// LS Electric XG5000 project: 주차설비
// PLC LSPLC
// module base 0 slot 0: 입출력 모듈:XBC-DN/DP64H (DC 24V 입력, 트랜지스터 출력 64점 (싱크출력/소스출력))

PROGRAM NewProgram (task: 스캔 프로그램)

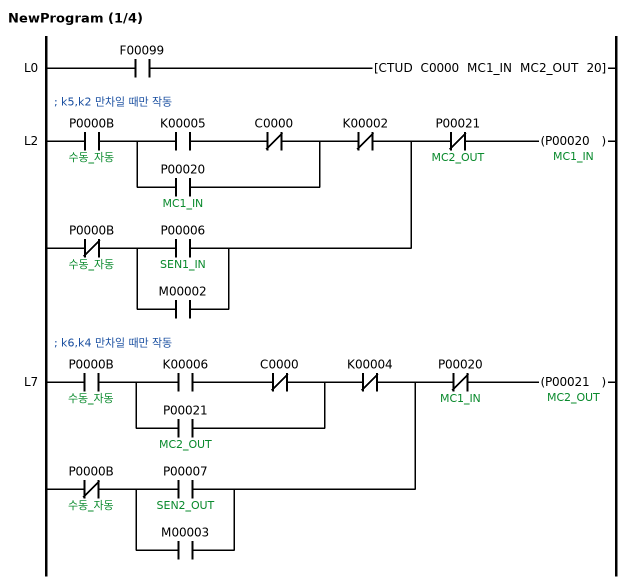
; L0
LOAD      F00099
CTUD      C0000 MC1_IN MC2_OUT 20
// k5,k2 만차일 때만 작동
; L2
LOAD      P0000B	// 수동_자동
LOAD      K00005
AND NOT   C0000
OR        P00020	// MC1_IN
AND LOAD
AND NOT   K00002
LOAD NOT  P0000B	// 수동_자동
LOAD      P00006	// SEN1_IN
OR        M00002
AND LOAD
OR LOAD
AND NOT   P00021	// MC2_OUT
OUT       P00020	// MC1_IN
// k6,k4 만차일 때만 작동
; L7
LOAD      P0000B	// 수동_자동
LOAD      K00006
AND NOT   C0000
OR        P00021	// MC2_OUT
AND LOAD
AND NOT   K00004
LOAD NOT  P0000B	// 수동_자동
LOAD      P00007	// SEN2_OUT
OR        M00003
AND LOAD
OR LOAD
AND NOT   P00020	// MC1_IN
OUT       P00021	// MC2_OUT

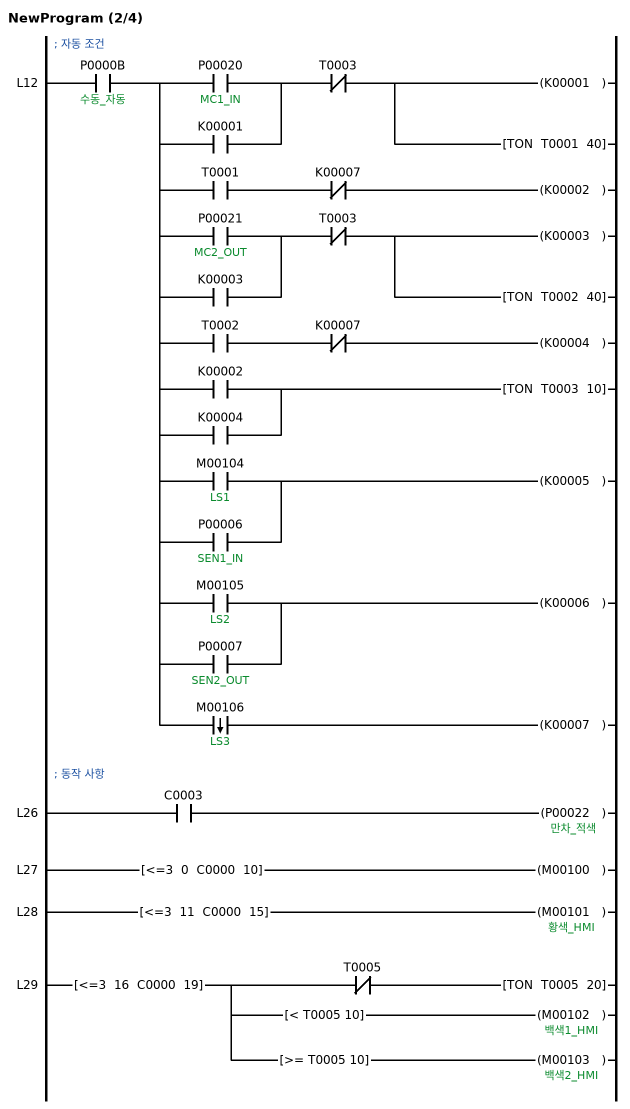
// 자동 조건
; L12
LOAD      P0000B	// 수동_자동
MPUSH
LOAD      P00020	// MC1_IN
OR        K00001
AND LOAD
AND NOT   T0003
OUT       K00001
TON       T0001 40
MLOAD
AND       T0001
AND NOT   K00007
OUT       K00002
MLOAD
LOAD      P00021	// MC2_OUT
OR        K00003
AND LOAD
AND NOT   T0003
OUT       K00003
TON       T0002 40
MLOAD
AND       T0002
AND NOT   K00007
OUT       K00004
MLOAD
LOAD      K00002
OR        K00004
AND LOAD
TON       T0003 10
MLOAD
LOAD      M00104	// LS1
OR        P00006	// SEN1_IN
AND LOAD
OUT       K00005
MLOAD
LOAD      M00105	// LS2
OR        P00007	// SEN2_OUT
AND LOAD
OUT       K00006
MPOP
ANDN      M00106	// LS3
OUT       K00007
// 동작 사항
; L26
LOAD      C0003
OUT       P00022	// 만차_적색
; L27
LOAD<=3   0 C0000 10
OUT       M00100
; L28
LOAD<=3   11 C0000 15
OUT       M00101	// 황색_HMI
; L29
LOAD<=3   16 C0000 19
MPUSH
AND NOT   T0005
TON       T0005 20
MLOAD
AND<      T0005 10
OUT       M00102	// 백색1_HMI
MPOP
AND>=     T0005 10
OUT       M00103	// 백색2_HMI

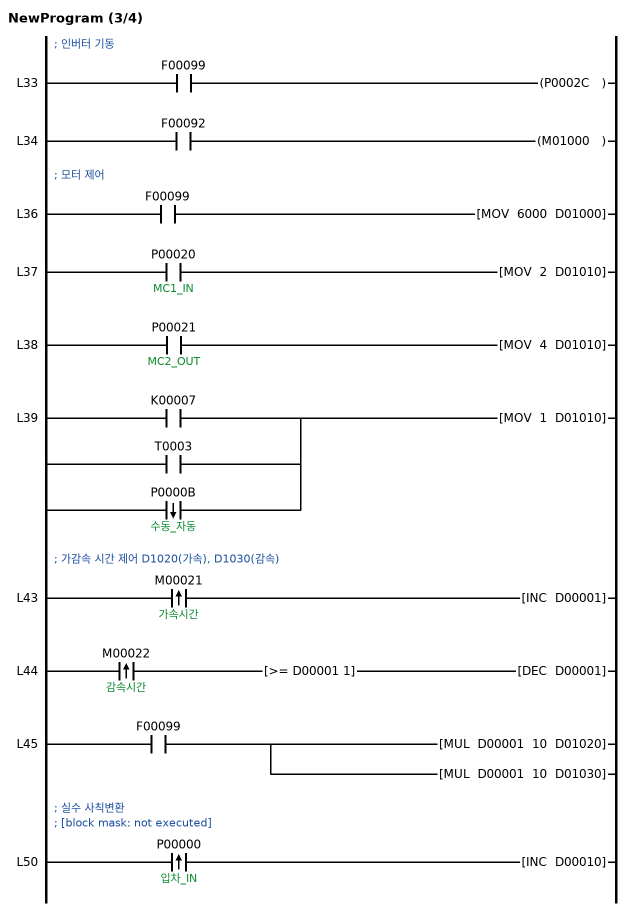
// 인버터 기동
; L33
LOAD      F00099
OUT       P0002C
; L34
LOAD      F00092
OUT       M01000
// 모터 제어
; L36
LOAD      F00099
MOV       6000 D01000
; L37
LOAD      P00020	// MC1_IN
MOV       2 D01010
; L38
LOAD      P00021	// MC2_OUT
MOV       4 D01010
; L39
LOAD      K00007
OR        T0003
ORN       P0000B	// 수동_자동
MOV       1 D01010
// 가감속 시간 제어 D1020(가속), D1030(감속)
; L43
LOADP     M00021	// 가속시간
INC       D00001
; L44
LOADP     M00022	// 감속시간
AND>=     D00001 1
DEC       D00001
; L45
LOAD      F00099
MUL       D00001 10 D01020
MUL       D00001 10 D01030
// 실수 사칙변환
; L50 (block mask: not executed)
LOADP     P00000	// 입차_IN
INC       D00010

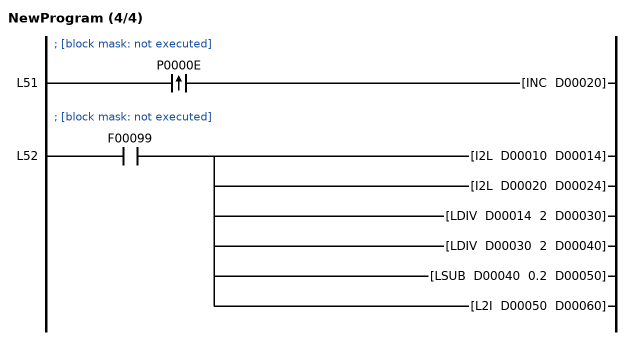
; L51 (block mask: not executed)
LOADP     P0000E
INC       D00020
; L52 (block mask: not executed)
LOAD      F00099
I2L       D00010 D00014
I2L       D00020 D00024
LDIV      D00014 2 D00030
LDIV      D00030 2 D00040
LSUB      D00040 0.2 D00050
L2I       D00050 D00060

VARIABLES AND COMMENTS (devices not used above)
M00200	BIT	녹색_HMI
P00001	BIT	출차_OUT